FUNCTION_BLOCK AIS_TO_AIS2 (* Composite FB for convert unidirectional AIS to bidirectional AIS2 *)
  (* Standard: 61499-2; Function: AIS_IN publishes its value onto the outgoing (EO1) side of AIS2_BIDIR. Whatever AIS2_BIDIR receives on its incoming (EI1) side is forwarded out again as a plain unidirectional signal via AIS_OUT.; Description: Copyright (c) 2026 HR Agrartechnik GmbH This program and the accompanying materials are made available under the terms of the Eclipse Public License 2.0 which is available at https://www.eclipse.org/legal/epl-2.0/ SPDX-License-Identifier: EPL-2.0 *)
  (* Version 1.0, 2026-09-12, Franz Höpfinger, HR Agrartechnik GmbH, Initial Version - Konvertierungsfamilie vervollstaendigt (analog zu AR2/AB2/AE2). *)
  PACKAGE adapter::conversion::bidirectional;
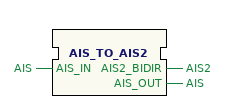
  SOCKETS
    AIS_IN : adapter::types::unidirectional::AIS; (* Adapter Input: unidirectional source *)
  END_SOCKETS
  PLUGS
    AIS2_BIDIR : adapter::types::bidirectional::AIS2; (* Adapter Output: bidirectional tap, outgoing side driven by AIS_IN, incoming side forwarded to AIS_OUT *)
    AIS_OUT : adapter::types::unidirectional::AIS; (* Adapter Output: mirrors AIS2_BIDIR's incoming (request) side *)
  END_PLUGS
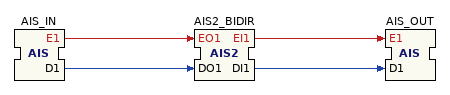
  EVENT_CONNECTIONS
    AIS_IN.E1 TO AIS2_BIDIR.EO1;
    AIS2_BIDIR.EI1 TO AIS_OUT.E1;
  END_CONNECTIONS
  DATA_CONNECTIONS
    AIS_IN.D1 TO AIS2_BIDIR.DO1;
    AIS2_BIDIR.DI1 TO AIS_OUT.D1;
  END_CONNECTIONS
END_FUNCTION_BLOCK
